FUNCTION_BLOCK ControlBlock
  (* Standard: 61499-2 *)
  (* Version 1.0, 2026-07-29, Dimitrios Kalligaridis *)
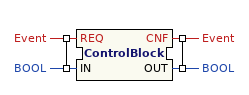
  EVENT_INPUT
    REQ WITH IN;
  END_EVENT
  EVENT_OUTPUT
    CNF WITH OUT;
  END_EVENT
  VAR_INPUT
    IN : BOOL;
  END_VAR
  VAR_OUTPUT
    OUT : BOOL;
  END_VAR
END_FUNCTION_BLOCK
